FUNCTION F_SetTransportTubeStatuses : BOOL
VAR_INPUT
	eTransportTube : T_TransportTube;
	stExpStatus : ST_TransportTubeStatuses;
	stStatusOp : ST_TransportTubeOps;
END_VAR
VAR
	fbTT : REFERENCE TO FB_TransportTube;
END_VAR

fbTT REF= F_GetTransportTube(eTransportTube);

IF NOT stStatusOp.bIonPumpIgnore THEN
	fbTT.q_stConfig.stDevices.refIonPump.M_Run(stExpStatus.bIonPumpOn);
END_IF
IF NOT stStatusOp.bGateValveIgnore THEN
	fbTT.q_stConfig.stDevices.refGateValve.M_Set_OPN_SW(stExpStatus.bGateValveOpen);
END_IF

END_FUNCTION

(* stored: Version 1.1.0.1, ProductVersion 3.1.4022.17
   POU F_SetTransportTubeStatuses: Id {71653e18-e337-4c05-b7ab-5fa8158795fd}, SpecialFunc None *)
